% RSLogix 500 project 02. Bar_Code_Reading_Registering.RSS, saved by version 8.30.00.16 %
PROJECT "UNTITLED"    % processor: Bul.1763 MicroLogix 1100 Series B %

PROGRAM FILES
  LAD 2 "MAIN"  6 rungs  % SISTEMA DE UM CÓDIGO DE BARRAS RECEBENDO STRING  %

DATA FILES
  O0 OUTPUT  4 elements
  I1 INPUT  6 elements
  S2 STATUS  66 elements
  B3 BINARY  1 elements
  T4 TIMER  1 elements
  C5 COUNTER  1 elements
  R6 CONTROL  1 elements
  N7 INTEGER  1 elements
  F8 FLOAT  1 elements
  ST9   6 elements
  ST10   1 elements

LADDER 2 "MAIN"    % SISTEMA DE UM CÓDIGO DE BARRAS RECEBENDO STRING  %
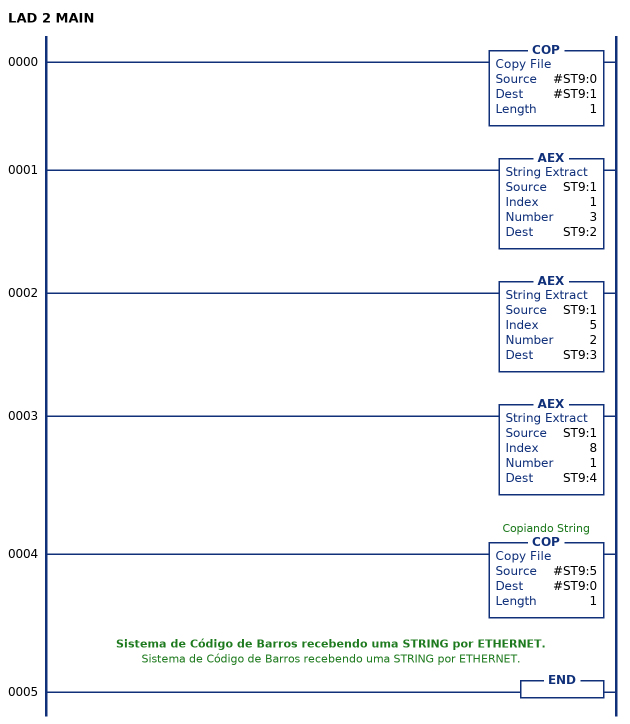
% Rung: 0 %
SOR COP #ST9:0 #ST9:1 1 EOR
%   ST9:0  "Copiando String" %
% Rung: 1 %
SOR AEX ST9:1 1 3 ST9:2 EOR
% Rung: 2 %
SOR AEX ST9:1 5 2 ST9:3 EOR
% Rung: 3 %
SOR AEX ST9:1 8 1 ST9:4 EOR
% Rung: 4 %
SOR COP #ST9:5 #ST9:0 1 EOR
%   ST9:5  ZERO %
%   ST9:0  "Copiando String" %
% Rung: 5 %
% TITLE: Sistema de Código de Barros recebendo uma STRING por ETHERNET. %
% Sistema de Código de Barros recebendo uma STRING por ETHERNET. %
SOR END EOR

DATA TABLE (non-zero values as saved)
DATA ST9
% ST9:2 % "789"
% ST9:3 % "05"
% ST9:4 % "2"
